(* Start/stop with a seal-in. Click StartPB > Force True, then Force False: Motor stays on. Click StopPB_NC > Force False to stop. *)

PROGRAM P1_StartStop
  VAR
    StartPB : BOOL; (* Start push-button, NO: TRUE while pressed *)
    StopPB_NC : BOOL := TRUE; (* Stop push-button, NC: TRUE while NOT pressed (a healthy stop circuit) *)
    Motor : BOOL; (* Motor contactor *)
    RunLamp : BOOL; (* Green running lamp *)
  END_VAR

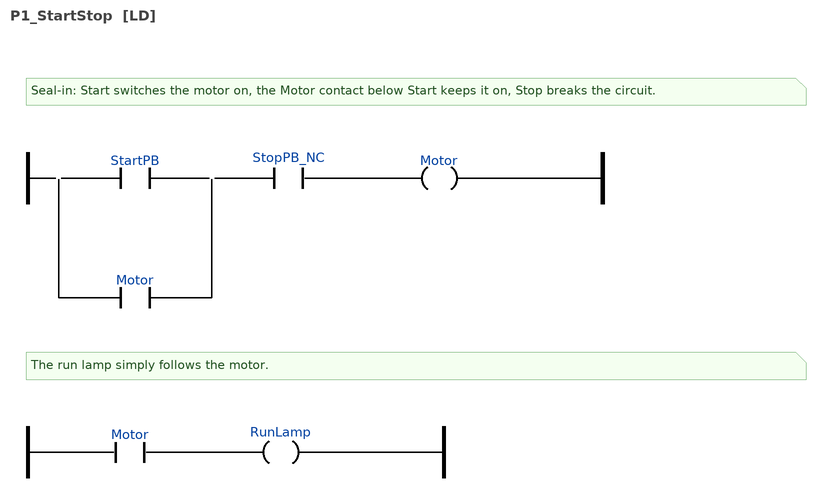
(* LD diagram, written out as Structured Text *)
(* Seal-in: Start switches the motor on, the Motor contact below Start keeps it on, Stop breaks the circuit. *)
Motor := (StartPB OR Motor) AND StopPB_NC;
(* The run lamp simply follows the motor. *)
RunLamp := Motor;
END_PROGRAM
